//Structure for specific subsystems related to an instrument --> MCC = one or more subysystems
TYPE ST_SubSystemOut :
STRUCT
END_STRUCT
END_TYPE

(* stored: Version 1.1.0.1
   DUT ST_SubSystemOut: Id {f647f3e9-2b7d-09a0-3ef9-d87937fd120b} *)
